// TIA Portal project "Proyecto3" (V16)

(* hardware
DEVICE "S7-1200 station_1"  S7-1200 Station
   slot 0: "Rack_0"  S7-1200 Rack  Rack  V1.0
   slot 1: "PLC_1"  CPU 1214C AC/DC/Rly  6ES7 214-1BG40-0XB0  V4.4
*)

// ===== PLC "PLC_1"  CPU 1214C AC/DC/Rly =====

VAR_GLOBAL   // PLC tag table "Tabla de variables estándar"
   ""Tag_1"" AT %I0.0 : Bool;
   ""Tag_2"" AT %I0.1 : Bool;
   ""Tag_3"" AT %Q0.0 : Bool;
END_VAR